FUNCTION_BLOCK FB_NotifyObserverAction EXTENDS FB_Action
VAR
    _pData: POINTER TO BYTE;
    _nSize: UDINT;
    _nTypeClass: __SYSTEM.TYPE_CLASS;
END_VAR

METHOD  Execute
VAR_INPUT
    ipObject: I_Object;
END_VAR
VAR
    ipObs: I_Observer;
END_VAR
__QUERYINTERFACE(ipObject, ipObs);

IF ipObs = 0 THEN
    RETURN;
END_IF

ipObs.UpdateP(pData := THIS^._pData,
              nTypeClass := THIS^._nTypeClass,
              nSize := THIS^._nSize);
END_METHOD

METHOD Inputs : I_Action
VAR_INPUT
    pData:          POINTER TO BYTE;
    nTypeClass:     __SYSTEM.TYPE_CLASS;
    nSize:          UDINT;
END_VAR
Inputs := THIS^;

THIS^._pData := pData;
THIS^._nTypeClass := nTypeClass;
THIS^._nSize := nSize;
END_METHOD

END_FUNCTION_BLOCK

(* stored: Version 1.1.0.1, ProductVersion 3.1.4024.12
   POU FB_NotifyObserverAction: Id {8cb99936-b569-4eab-bcc8-0631bace8fa9}, SpecialFunc None
   Method Execute: Id {87f751f9-c536-4b1f-996b-5ae96ee166a6}
   Method Inputs: Id {f57e0d64-abd4-42b5-8230-4dbde712a3ff} *)
